// TwinCAT 3 PLC project PLC1
// ProgramVersion: 3.1.4024.0
// libraries:
//   Tc2_MC2, * (Beckhoff Automation GmbH)
//   Tc2_NcKinematicTransformation, * (Beckhoff Automation GmbH)
//   Tc2_Standard, * (Beckhoff Automation GmbH)
//   Tc2_System, * (Beckhoff Automation GmbH)
//   Tc3_Module, * (Beckhoff Automation GmbH)
// project tree:
//   / PlcTask.TcTTO
//   POUs/ MAIN.TcPOU
// real-time tasks:
//   TASK PlcTask: cycle T#10ms, priority 20, ADS port 350
// motion (NC):
//   TASK NC-Task 1 SAF: cycle T#2ms, priority 4, ADS port 501
//   TASK NC-Task 1 SVB: cycle T#10ms, priority 8, ADS port 511
//   AXIS X (id 5)
//     OtherSettings: AllowMotionCmdToSlave=true
//     encoder EncType=1
//     drive DrvType=5
//       Analog: TorqueSetpointScale=10, ScaleFactorActTorque=0.1
//     controller CtrType=1
//       CtrPara: PriorControlFactor=1
//         Observer: BandWidth=20
//   AXIS Y (id 6)
//   AXIS Z (id 7)
//   AXIS C (id 8)
//   AXIS Axis 1 (id 1)
//   AXIS Axis 2 (id 2)
//     OtherSettings: AllowMotionCmdToSlave=true
//     encoder EncType=1
//     drive DrvType=5
//       Analog: TorqueSetpointScale=10, ScaleFactorActTorque=0.1
//     controller CtrType=1
//       CtrPara: PriorControlFactor=1
//         Observer: BandWidth=20
//   AXIS Axis 3 (id 3)
//   AXIS Axis 4 (id 4)
// variable links:
//   PLC1 Instance <-> NC-Task 1 SAF/Axes/Axis 1
//     PlcTask Inputs/MAIN.ACS_Axis[1].NcToPlc <-> Outputs/ToPlc
//     PlcTask Outputs/MAIN.ACS_Axis[1].PlcToNc <-> Inputs/FromPlc
//   PLC1 Instance <-> NC-Task 1 SAF/Axes/Axis 2
//     PlcTask Inputs/MAIN.ACS_Axis[2].NcToPlc <-> Outputs/ToPlc
//     PlcTask Outputs/MAIN.ACS_Axis[2].PlcToNc <-> Inputs/FromPlc
//   PLC1 Instance <-> NC-Task 1 SAF/Axes/Axis 3
//     PlcTask Inputs/MAIN.ACS_Axis[3].NcToPlc <-> Outputs/ToPlc
//     PlcTask Outputs/MAIN.ACS_Axis[3].PlcToNc <-> Inputs/FromPlc
//   PLC1 Instance <-> NC-Task 1 SAF/Axes/Axis 4
//     PlcTask Inputs/MAIN.ACS_Axis[4].NcToPlc <-> Outputs/ToPlc
//     PlcTask Outputs/MAIN.ACS_Axis[4].PlcToNc <-> Inputs/FromPlc
//   PLC1 Instance <-> NC-Task 1 SAF/Axes/C
//     PlcTask Inputs/MAIN.MCS_Axis[4].NcToPlc <-> Outputs/ToPlc
//     PlcTask Outputs/MAIN.MCS_Axis[4].PlcToNc <-> Inputs/FromPlc
//   PLC1 Instance <-> NC-Task 1 SAF/Axes/X
//     PlcTask Inputs/MAIN.MCS_Axis[1].NcToPlc <-> Outputs/ToPlc
//     PlcTask Outputs/MAIN.MCS_Axis[1].PlcToNc <-> Inputs/FromPlc
//   PLC1 Instance <-> NC-Task 1 SAF/Axes/Y
//     PlcTask Inputs/MAIN.MCS_Axis[2].NcToPlc <-> Outputs/ToPlc
//     PlcTask Outputs/MAIN.MCS_Axis[2].PlcToNc <-> Inputs/FromPlc
//   PLC1 Instance <-> NC-Task 1 SAF/Axes/Z
//     PlcTask Inputs/MAIN.MCS_Axis[3].NcToPlc <-> Outputs/ToPlc
//     PlcTask Outputs/MAIN.MCS_Axis[3].PlcToNc <-> Inputs/FromPlc
//   PLC1 Instance <-> NC-Task 1 SAF/Kin_Trafo_Channel
//     PlcTask Inputs/MAIN.in_stKinToPlc <-> Outputs/ToPlc
//     PlcTask Outputs/MAIN.out_stPlcToKin <-> Inputs/FromPlc

CONFIGURATION PLC1
    RESOURCE PLC ON TwinCAT3
        TASK PlcTask(INTERVAL := T#10ms, PRIORITY := 20);
        PROGRAM MAIN WITH PlcTask : MAIN;
    END_RESOURCE
END_CONFIGURATION

// ---- POUs/MAIN.TcPOU
PROGRAM MAIN
VAR	
	{region 'NC Variables'}
	// Status Array of MCS Position
	MCS_Positions : ARRAY[1..MAX_MCS_AXES] OF LREAL;	
	// Axis Control Ref for ACS
	ACS_Axis		: ARRAY[1..MAX_ACS_AXES] OF Axis_Ref;
	// Axis Control Ref for MCS
	MCS_Axis		: ARRAY[1..MAX_MCS_AXES] OF Axis_Ref;
	// ACS Axis Power Block
	mcACS_Power 	: ARRAY[1..MAX_ACS_AXES] OF MC_Power;
	// MCS Axis Power Block
	mcMCS_Power 	: ARRAY[1..MAX_MCS_AXES] OF MC_Power;
	// Axis Set Position Block
	mcSetPosition 	: ARRAY[1..MAX_ACS_AXES] OF MC_SetPosition;
	{endregion}
		 
	{region  'Kinematics Variables'}
	// Kinematic Model Reference
	{attribute 'TcInitSymbol'}
	oidTrafo			: OTCID;
	// Struct In from Kin Channel
	in_stKinToPlc      AT %I*     : NCTOPLC_NCICHANNEL_REF;
	// Struct Out to Kin Channel
	out_stPlcToKin     AT %Q*     : PLCTONC_NCICHANNEL_REF;	 
	// Axes Configuration Structure
	stAxesConfig		: ST_KinAxes;
	// Kinematics Configuration Group			  
	fbConfigKinGroup	: FB_KinConfigGroup;
	// Reset the Kin Group
	fbResetKinGroup   : FB_KinResetGroup;
	// Calculating the Trafo
	fbKinCalcTrafo		: FB_KinCalcTrafo;
	// Struct of position into the calculation
    stAxesPosIn			: ARRAY[1..8] OF LREAL;
	// Struct of positions out
    stAxesPosOut		: ARRAY[1..8] OF LREAL;			  
	// Scara Meta Info 
	uScaraMetaInfoIn	: U_KinMetaInfo;
	// Scara Meta Info
    uScaraMetaInfoOut	: U_KinMetaInfo;
  	// Unlock Trafo
	fbUnlockTrafoParam	: FB_KinUnlockTrafoParam;
	// Lock Trafo
	fbLockTrafoParam	: FB_KinLockTrafoParam;
	// ADS Write Block
    fbADSWRITE			: ADSWRITE;	
	// Parameter ID to Change (*Inner Arm Length*)
	pidTrafo			: UDINT := 16#05010020; 
	// Value to write to the parameter
	fParamValue			: LREAL := 400.0;			  
	{endregion}

	{region  'General System Variables'}
	// Loop Iterator
	I_itr			: INT;
	{endregion}
		 
	{region 'State Machine Variables'}
	// State of the state machine
	nState 			: INT;
	// Control Variables
	bStart, bHalt 	: BOOL;
	// Control the steps
	bStep1, bFixStep, bStep2, bStep3, bStep4, bStep5, bStep6 : BOOL;
	{endregion}
END_VAR
VAR CONSTANT
	{region  'Axes Constants'}
	// ACS Axes Count
	MAX_ACS_AXES 		: INT := 4;
	// MCS Axes Count
	MAX_MCS_AXES 		: INT := 4;
	// Joint Positions
	AXES_JOINT_POSE	: ARRAY[1..MAX_ACS_AXES] OF LREAL := [0.0, 90.0, 0.0, 0.0];
	{endregion}
END_VAR

// Simple NC State Machine

CASE nState OF
	{region 'Start of State Machine'}
	0:	// Start the state machine
		IF bStart THEN
			bStart := FALSE;
			nState := nState + 10;
		END_IF
	{endregion}
	
	{region 'ACS Power Section'}
	10: // Power on the axis
		FOR I_itr := 1 TO MAX_ACS_AXES DO
			mcACS_Power[I_itr](Axis := ACS_Axis[I_itr], Enable := TRUE, Enable_Positive := TRUE, Enable_Negative := TRUE, Override := 100.0);
		END_FOR
		nState := nState + 10;
	
	20: // Check all axis are enabled
		FOR I_itr := 1 TO MAX_ACS_AXES DO
			// Check if motor is enabled
			IF NOT mcACS_Power[I_itr].Status THEN
				// Return to power state, or reset state if you have one
				// At the end of this state we add 10, so to return to 10 we need to subtract 20
				nState := nState - 20;
				EXIT;
			END_IF
		END_FOR
		nState := nState + 10;
	{endregion}
		 
	{region 'MCS Power Section'}
	30: // Power on the axis
		FOR I_itr := 1 TO MAX_MCS_AXES DO
			mcMCS_Power[I_itr](Axis := MCS_Axis[I_itr], Enable := TRUE, Enable_Positive := TRUE, Enable_Negative := TRUE, Override := 100.0);
		END_FOR
		nState := nState + 10;
	
	40: // Check all axis are enabled
		FOR I_itr := 1 TO MAX_MCS_AXES DO
			// Check if motor is enabled
			IF NOT mcMCS_Power[I_itr].Status THEN
				// Return to power state, or reset state if you have one
				// At the end of this state we add 10, so to return to 10 we need to subtract 20
				nState := nState - 20;
				EXIT;
			END_IF
		END_FOR
		nState := nState + 10;
	{endregion}

	{region 'Starting point for steps'}
	50: // Wait State
		IF bStep1 THEN
			bStep1 := FALSE;
			nState := nState + 10;
		END_IF
	{endregion}
	  
	{region 'Step 1 - Assemble the Axes List Struct'}	
	60: (*
		**	Step 1 - Assemble the Axes List Struct
		*)
		(*******************************************)
		// Assign the ACS Axes
		FOR I_itr := 1 TO MAX_ACS_AXES DO
			stAxesConfig.nAxisIdsAcs[I_itr] := ACS_Axis[I_itr].NcToPlc.AxisId;
	 	END_FOR
		// Assign the MCS Axes
		FOR I_itr := 1 TO MAX_MCS_AXES DO
			stAxesConfig.nAxisIdsMcs[I_itr] := MCS_Axis[I_itr].NcToPlc.AxisId;
	 	END_FOR
		(*******************************************)
		IF bFixStep	THEN
			nState := nState + 10; 		 
		END_IF	
	{endregion}
		 
	{region 'Step 2 - Fixing Issues}
	70:	// Step 2 might have an issue, here is where you'll fix it
		(**********************************************************)
		FOR I_itr := 1 TO MAX_ACS_AXES DO
			mcSetPosition[I_itr](Axis := ACS_Axis[I_itr], Execute := TRUE, Position := AXES_JOINT_POSE[I_itr]);		 
	 	END_FOR
		(**********************************************************)	 
		nState := nState + 10; 
			 
	80: // Check if the command is complete
		(**********************************************************)
		FOR I_itr := 1 TO MAX_ACS_AXES DO
			mcSetPosition[I_itr](Axis := ACS_Axis[I_itr], Execute := FALSE, Position := AXES_JOINT_POSE[I_itr]);		 
	 	END_FOR
		(**********************************************************)	 
		IF bStep2 THEN
			bStep2 := FALSE;
			nState := nState + 10;
		END_IF		 
	{endregion}
		 
	{region 'Step 2 - Configure Kinematic Group'}		 
	90: (*
		**	Step 2 - Configure Kinematic Group
		*)
		(*******************************************)
		fbConfigKinGroup(bExecute := TRUE, bCartesianMode := TRUE, stAxesList := stAxesConfig, stKinRefIn := in_stKinToPlc); 
		// If you get an error, think about why it doesnt work
		IF fbConfigKinGroup.bDone THEN
			nState := nState + 10;	 
		END_IF
		(*******************************************)					   
	{endregion}	
		 		  	 
	{region 'Step 3 - Move the configuration'}		
	100: (*
		** Step 3 - Move the configuration
		*)
		(*******************************************	 
		*******************************************)					   
		IF bStep5 THEN
			bStep5 := FALSE;
			nState := nState + 10;
		END_IF
	{endregion}
		
	{region 'Step 5 - Break the Kinematic Group'}	
	110: (*
		** Step 5 - Break the Kinematic Group
		** NOTE : Step 4 is at the bottom of POU
		*)
		(*******************************************)
		fbResetKinGroup(
			bExecute := TRUE, 
			nItpChannelId := in_stKinToPlc.ChnId, 
			stKinRefIn := in_stKinToPlc, 
			stAxesList := stAxesConfig);
				 
		IF fbResetKinGroup.bDone THEN
			fbResetKinGroup(bExecute := FALSE, nItpChannelId := in_stKinToPlc.ChnId, stKinRefIn := in_stKinToPlc, stAxesList := stAxesConfig);	 
			nState := nState + 10;	 
		END_IF		 
		(*******************************************)					   
	{endregion}
		 
	{region 'Wait state before Step 6'}
	120: // Wait state before step 6
		IF bStep6 THEN
			bStep6 := FALSE;
			nState := nState + 10;
		END_IF
	{endregion}
	
	{region 'Step 6 - Unlock Trafo and Modify Params'}		
	130: (*
		** Step 6 - Unlock Trafo and Modify Params
		*)
		(*******************************************)
		fbUnlockTrafoParam(bExecute := TRUE, oidTrafo := oidTrafo);
		IF fbUnlockTrafoParam.bDone THEN
			fbUnlockTrafoParam(bExecute := FALSE, oidTrafo := oidTrafo);
			nState := nState + 10;	 
		END_IF
			 
	140: // Write the value with ADS
		fbADSWRITE(	NETID:='' ,
					PORT:= AMSPORT_R0_NCSAF,
					IDXGRP:=oidTrafo ,
					IDXOFFS:= pidTrafo,
					LEN:=SIZEOF(fParamValue) ,
					SRCADDR:= ADR(fParamValue),
					WRITE:=TRUE);	

		IF NOT fbADSWRITE.BUSY THEN
			fbADSWRITE(WRITE:=FALSE);
			nState := nState + 10;	 
		END_IF	  
		
	150: // Lock Trafo back up
		fbLockTrafoParam(bExecute := TRUE, oidTrafo := oidTrafo);					   
		IF fbLockTrafoParam.bDone THEN
			fbLockTrafoParam(bExecute := FALSE, oidTrafo := oidTrafo);
			nState := nState + 10;
		END_IF
		(*******************************************)		 
	{endregion}
		
	{region 'End of State Machine'}
	160: // Check if continuous loop, or return to 0
		IF bStep1 THEN
			bStep1 := FALSE;
			nState := 60;
		END_IF
	{endregion}		
END_CASE

{region 'Step 4 - Calculate the Transformation'}	
(* 
** Step 4 - Calculate the Transformation
*)
IF bStep4 THEN
(***********************************************)
	// Toggle eveything false		 
	fbKinCalcTrafo(
		bExecute := FALSE,	
		bForward := FALSE, 
		stAxesPosIn := stAxesPosIn, 
		stAxesPosOut := stAxesPosOut, 
		uMetaInfoIn:= uScaraMetaInfoIn, 
		uMetaInfoOut:= uScaraMetaInfoOut);
		 
	// Check if Kinematics is running, if not then calculate the MCS
	IF F_KinGetChnOperationState(stKinRefIn := in_stKinToPlc) = E_KinStatus.KinStatus_Ready THEN
		FOR I_itr := 1 TO MAX_MCS_AXES DO
			MCS_Positions[I_itr] := MCS_Axis[I_itr].NcToPlc.ActPos;
		END_FOR		 
	ELSE
		// Copy the ACS positions for calculation
		FOR I_itr := 1 TO MAX_MCS_AXES DO
			stAxesPosIn[I_itr] := ACS_Axis[I_itr].NcToPlc.ActPos;
		END_FOR		 
		// Tell the calculation that the SCARA is a Right Arm		  
		uScaraMetaInfoIn.eScara := E_KinMetaInfoScara.scaraRightArm;
		
		// Compute the kinematics
		fbKinCalcTrafo(
			bExecute := TRUE, 
			bForward := TRUE, 
			oidTrafo := oidTrafo, 
			stAxesPosIn := stAxesPosIn, 
			stAxesPosOut := stAxesPosOut, 
			uMetaInfoIn:= uScaraMetaInfoIn, 
			uMetaInfoOut:= uScaraMetaInfoOut); 	
				 
		// Copy the computed values into the MCS_Position array
		FOR I_itr := 1 TO MAX_MCS_AXES DO
			MCS_Positions[I_itr] := stAxesPosOut[I_itr];
		END_FOR	
			  
	END_IF
(***********************************************)
END_IF
{endregion}

END_PROGRAM
